{attribute 'qualified_only'}
VAR_GLOBAL
	// ingressi
	start: BOOL;
	stop : BOOL;
	emg  : BOOL;
	ack  : BOOL;
	fc1  : BOOL;
	fc2  : BOOL;
	
	// uscite
	H1   : BOOL;
	HEMG : BOOL;
	M    : BOOL;
	// il nastro è libero
	libero : BOOL; 	
END_VAR

(* stored: Version 1.1.0.1
   GVL GVL_IO: Id {ee47021c-7c45-0f7d-05d3-ab9b71e08a51} *)
